// TIA Portal V20 export
// export: Created 2026-04-11T06:02:30.8208567Z, ExportSetting WithDefaults, DisplayName Totally Integrated Automation Portal, DisplayVersion V20, DisplayName TIA Portal Openness, DisplayVersion V20, DisplayName TIA Portal Version Control Interface, DisplayVersion V20, DisplayName STEP 7 Professional, DisplayVersion V20, DisplayName STEP 7 Safety, DisplayVersion V20, DisplayName WinCC Basic/Comfort/Advanced, DisplayVersion V20, DisplayName WinCC Unified, DisplayVersion V20
TYPE "mb_station_block_udt"
// stored: IsFailsafeCompliant false
   STRUCT
      conf : Struct   // Configuration
         skip_code : Bool;
         disable { S7_SetPoint := 'True'} : Bool;   // Skip all queries
         read_only { S7_SetPoint := 'True'} : Bool;   // Skip all write queries. (fc 5,6,15,16)
         max_comm_error { S7_SetPoint := 'True'} : USInt := 2;   // Repeating erros before communication_error flag is set
         exec_x_quries { S7_SetPoint := 'True'} : USInt := 1;   // Number of queries to be exec. at each loop.
      END_STRUCT;
      out { ExternalWritable := 'False'} : Struct   // Outputs
         error { ExternalWritable := 'False'} : Bool;   // All errors, including communication errors
         error_comm { ExternalWritable := 'False'} : Bool;   // only communication errors
         finnish { ExternalWritable := 'False'} : Bool;   // qid is handed over to next device.
      END_STRUCT;
      log { ExternalWritable := 'False'} : Struct   // Logging for development and debugging.
         connected_time { ExternalWritable := 'False'} : DTL;   // The time the device was connected to the bus
         disconnected_time { ExternalWritable := 'False'} : DTL;   // The time, if a device was disconnected to the bus
         done_cnt { ExternalWritable := 'False'} : UDInt;   // Successfully queries counter for this device
         error_comm_cnt { ExternalWritable := 'False'} : UDInt;   // Communication erros cnt.
         error_exception_cnt { ExternalWritable := 'False'} : UDInt;   // Failed queries counter for this device
         error_status { ExternalWritable := 'False'} : Word;   // Status code from mb_master or mb_client
         error_data_addr { ExternalWritable := 'False'} : UDInt;   // d_addr for last failed querie; handy for troubleshooting
      END_STRUCT;
      z { ExternalAccessible := 'False'; ExternalVisible := 'False'; ExternalWritable := 'False'} : Struct   // Internal states.
         header_qid { ExternalAccessible := 'False'; ExternalVisible := 'False'; ExternalWritable := 'False'} : UInt;   // qid value at device header
         comm_err_cnt { ExternalAccessible := 'False'; ExternalVisible := 'False'; ExternalWritable := 'False'} : USInt;   // Repeating communication errors
         exec_cnt { ExternalAccessible := 'False'; ExternalVisible := 'False'; ExternalWritable := 'False'} : USInt;   // Numb. of exec. q. this loop
         offset_qid { ExternalAccessible := 'False'; ExternalVisible := 'False'; ExternalWritable := 'False'} : UInt := 1;   // Device query id.
         err_hold { ExternalAccessible := 'False'; ExternalVisible := 'False'; ExternalWritable := 'False'} : Bool;   // Help var for .out.error
      END_STRUCT;
   END_STRUCT;
END_TYPE
